{attribute 'GeneratedUsingTerminal: EL4038-0000-0016'}
{attribute addProperty BoxType "EL4038-0000-0016"}
{attribute addProperty Id "AO_Outputs_Channel_1AT %Q*AO_Outputs_Channel_BA7EBB7C2AO_Outputs_Channel_2AT %Q*AO_Outputs_Channel_BA7EBB7C2AO_Outputs_Channel_3AT %Q*AO_Outputs_Channel_BA7EBB7C2AO_Outputs_Channel_4AT %Q*AO_Outputs_Channel_BA7EBB7C2AO_Outputs_Channel_5AT %Q*AO_Outputs_Channel_BA7EBB7C2AO_Outputs_Channel_6AT %Q*AO_Outputs_Channel_BA7EBB7C2AO_Outputs_Channel_7AT %Q*AO_Outputs_Channel_BA7EBB7C2AO_Outputs_Channel_8AT %Q*AO_Outputs_Channel_BA7EBB7C2WcStateAT %I*WcState_0B2B16F91InfoDataAT %I*InfoData_94A18F5E2"}
{attribute addProperty CRC "626604214"}
{attribute addProperty Size "19"}
TYPE EL4038_255938B6 EXTENDS EtcSlaveTerminalBase_947E5A46 :
STRUCT
	{attribute addProperty Name "AO_Outputs_Channel_1"}
	AO_Outputs_Channel_1 : AO_Outputs_Channel_BA7EBB7C;
	{attribute addProperty Name "AO_Outputs_Channel_2"}
	AO_Outputs_Channel_2 : AO_Outputs_Channel_BA7EBB7C;
	{attribute addProperty Name "AO_Outputs_Channel_3"}
	AO_Outputs_Channel_3 : AO_Outputs_Channel_BA7EBB7C;
	{attribute addProperty Name "AO_Outputs_Channel_4"}
	AO_Outputs_Channel_4 : AO_Outputs_Channel_BA7EBB7C;
	{attribute addProperty Name "AO_Outputs_Channel_5"}
	AO_Outputs_Channel_5 : AO_Outputs_Channel_BA7EBB7C;
	{attribute addProperty Name "AO_Outputs_Channel_6"}
	AO_Outputs_Channel_6 : AO_Outputs_Channel_BA7EBB7C;
	{attribute addProperty Name "AO_Outputs_Channel_7"}
	AO_Outputs_Channel_7 : AO_Outputs_Channel_BA7EBB7C;
	{attribute addProperty Name "AO_Outputs_Channel_8"}
	AO_Outputs_Channel_8 : AO_Outputs_Channel_BA7EBB7C;
	{attribute addProperty Name "WcState"}
	WcState : WcState_0B2B16F9;
	{attribute addProperty Name "InfoData"}
	InfoData : InfoData_94A18F5E;
END_STRUCT
END_TYPE

(* stored: Version 1.2.0.0, ProductVersion 3.1.4024.9
   DUT EL4038_255938B6: Id {2ca1dc6c-2a1a-4373-9c27-84b13fd24214} *)
